// TIA Portal V17 export
// export: Created 2025-06-26T07:49:40.7746535Z, ExportSetting WithDefaults, DisplayName Totally Integrated Automation Portal, DisplayVersion V17 Update 8, DisplayName TIA Portal Openness, DisplayVersion V17 Update 8, DisplayName TIA Portal Version Control Interface, DisplayVersion V17, DisplayName STEP 7 Professional, DisplayVersion V17 Update 8, DisplayName STEP 7 Safety, DisplayVersion V17 Update 6, DisplayName WinCC Advanced, DisplayVersion V17 Update 8
FUNCTION_BLOCK "Evaluate"   // FB26, FBD
TITLE = Evaluate machine state conditions
{ S7_Optimized_Access := 'TRUE' }
AUTHOR : Heaten
VERSION : 0.1
// stored: AutoNumber true, IsIECCheckEnabled false, IsRetainMemResEnabled false, MemoryReserve 0, SetENOAutomatically false, UDAEnableTagReadback false
   VAR
      TOF2_StandbyPauseTime { S7_SetPoint := 'True'} : TOF_TIME;
      TON2_Standby { S7_SetPoint := 'True'} : TON_TIME;
      TON3_PrepareStart { S7_SetPoint := 'True'} : TON_TIME;
      TON4_Start { S7_SetPoint := 'True'} : TON_TIME;
      TON5_Warmup { S7_SetPoint := 'True'} : TON_TIME;
      TON7_Stop { S7_SetPoint := 'True'} : TON_TIME;
      MinimumPriming { S7_SetPoint := 'True'} : TON_TIME;
   END_VAR
   VAR_TEMP
      HydrolockSpeed : Real;
      HeatSinkTemperatureMax : Real;
   END_VAR
BEGIN

REGION Network 1: Check running condition: system initialized
   // Add more conditions here
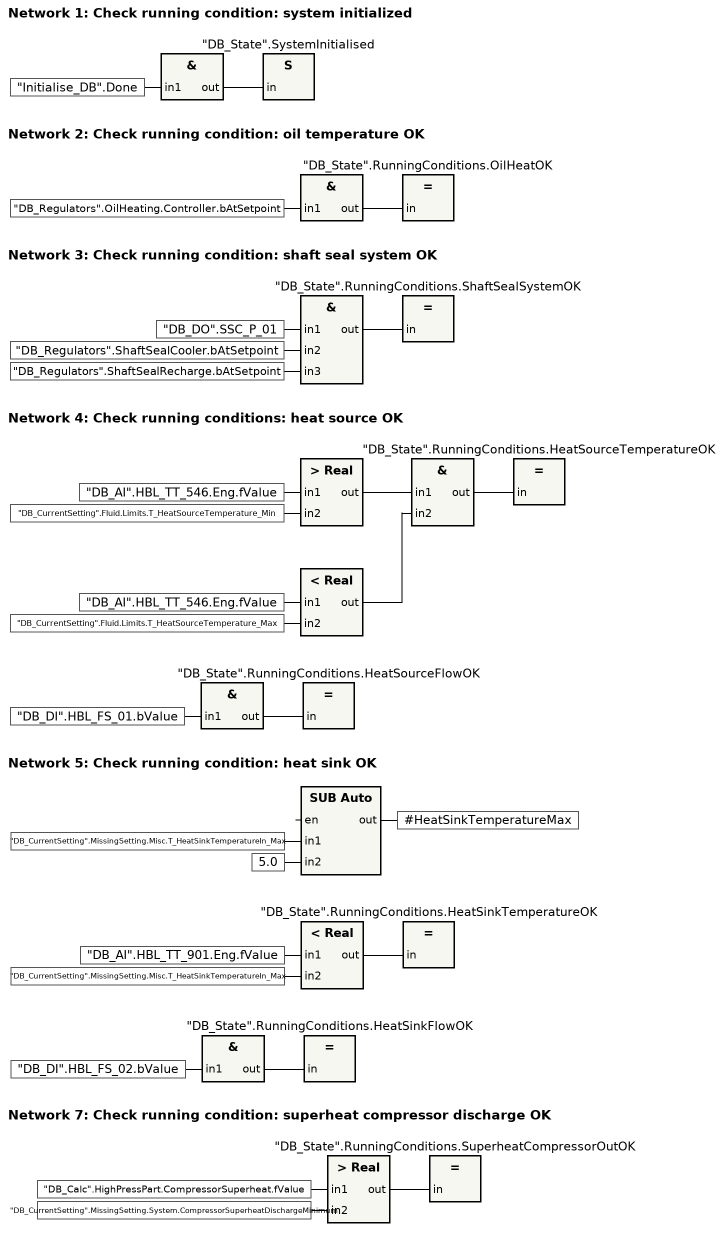
   IF "Initialise_DB".Done THEN "DB_State".SystemInitialised := TRUE; END_IF;
END_REGION

REGION Network 2: Check running condition: oil temperature OK
   "DB_State".RunningConditions.OilHeatOK := "DB_Regulators".OilHeating.Controller.bAtSetpoint;
END_REGION

REGION Network 3: Check running condition: shaft seal system OK
   "DB_State".RunningConditions.ShaftSealSystemOK := "DB_DO".SSC_P_01 AND "DB_Regulators".ShaftSealCooler.bAtSetpoint AND "DB_Regulators".ShaftSealRecharge.bAtSetpoint;
END_REGION

REGION Network 4: Check running conditions: heat source OK
   "DB_State".RunningConditions.HeatSourceTemperatureOK := ("DB_AI".HBL_TT_546.Eng.fValue > "DB_CurrentSetting".Fluid.Limits.T_HeatSourceTemperature_Min) AND ("DB_AI".HBL_TT_546.Eng.fValue < "DB_CurrentSetting".Fluid.Limits.T_HeatSourceTemperature_Max);
   "DB_State".RunningConditions.HeatSourceFlowOK := "DB_DI".HBL_FS_01.bValue;
END_REGION

REGION Network 5: Check running condition: heat sink OK
   // NOTE: leave a little headroom to the limit for standby, otherwise the machine shuts down (via alarm 2101) at the same temperature as it should go to standby on
   #HeatSinkTemperatureMax := "DB_CurrentSetting".MissingSetting.Misc.T_HeatSinkTemperatureIn_Max - 5.0;
   "DB_State".RunningConditions.HeatSinkTemperatureOK := "DB_AI".HBL_TT_901.Eng.fValue < "DB_CurrentSetting".MissingSetting.Misc.T_HeatSinkTemperatureIn_Max;
   "DB_State".RunningConditions.HeatSinkFlowOK := "DB_DI".HBL_FS_02.bValue;
END_REGION

REGION Network 6 (SCL): Check running condition: recuperator working
   // Recuperator sits between evaporator and compressor and SHOULD INCREASE THE SUPERHEAT (ie delta T over the recuperator should be positive)
   // 
   // Recuperator window: must add at least "DB_CurrentSetting".MissingSetting.System.RecuperatorSuperheatGainWorking degrees to be considered working, 
   // but can then fall as low as "DB_CurrentSetting".MissingSetting.System.RecuperatorSuperheatGainNotWorking degrees before it is considered not working again
   (*
   IF ("DB_Calc".LowPressPart.CompressorSuperheat.fValue - 2) <      //If the superheat at compressor inlet minus 2 is smaller than
       "DB_Calc".LowPressPart.EvaporatorSuperheat.fValue THEN          //the superheat at the evaporator, the recuperator doesn´t work
       "StateMachine_DB".RunningConditions.RecuperatorWorking := FALSE;
   ELSIF
       ("DB_Calc".LowPressPart.CompressorSuperheat.fValue + 3) >     //If the superheat at compressor inlet plus 3 is bigger than
       "DB_Calc".LowPressPart.EvaporatorSuperheat.fValue THEN          //the superheat at the evaporator, the recuperator works
       "StateMachine_DB".RunningConditions.RecuperatorWorking := TRUE;
   END_IF;
   *)

   // Rewritten with user-defined limits and right-side-up logic
   // Also don't evaluate the condition unless it's relevant, to avoid odd conditions during earlier states/cold start setting this accidentally
   IF "DB_State".State.State_Number = 5 OR "DB_State".State.State_Number = 6 THEN
       IF "DB_Calc".LowPressPart.CompressorSuperheat.fValue > "DB_Calc".LowPressPart.EvaporatorSuperheat.fValue + "DB_CurrentSetting".MissingSetting.System.RecuperatorDeltaTWorking THEN
           "DB_State".RunningConditions.RecuperatorWorking := TRUE;
       ELSIF "DB_Calc".LowPressPart.CompressorSuperheat.fValue < "DB_Calc".LowPressPart.EvaporatorSuperheat.fValue + "DB_CurrentSetting".MissingSetting.System.RecuperatorDeltaTNotWorking THEN
           "DB_State".RunningConditions.RecuperatorWorking := FALSE;
       END_IF;
   ELSE
       "DB_State".RunningConditions.RecuperatorWorking := FALSE;
   END_IF;
END_REGION

REGION Network 7: Check running condition: superheat compressor discharge OK
   "DB_State".RunningConditions.SuperheatCompressorOutOK := "DB_Calc".HighPressPart.CompressorSuperheat.fValue > "DB_CurrentSetting".MissingSetting.System.CompressorSuperheatDischargeMinimum;
END_REGION

REGION Network 8: Check running condition: at or above hydrolock speed
   // Give a small margin for error, so if it sits at, for example 288.2 RPM and the limit is 290, it will work.
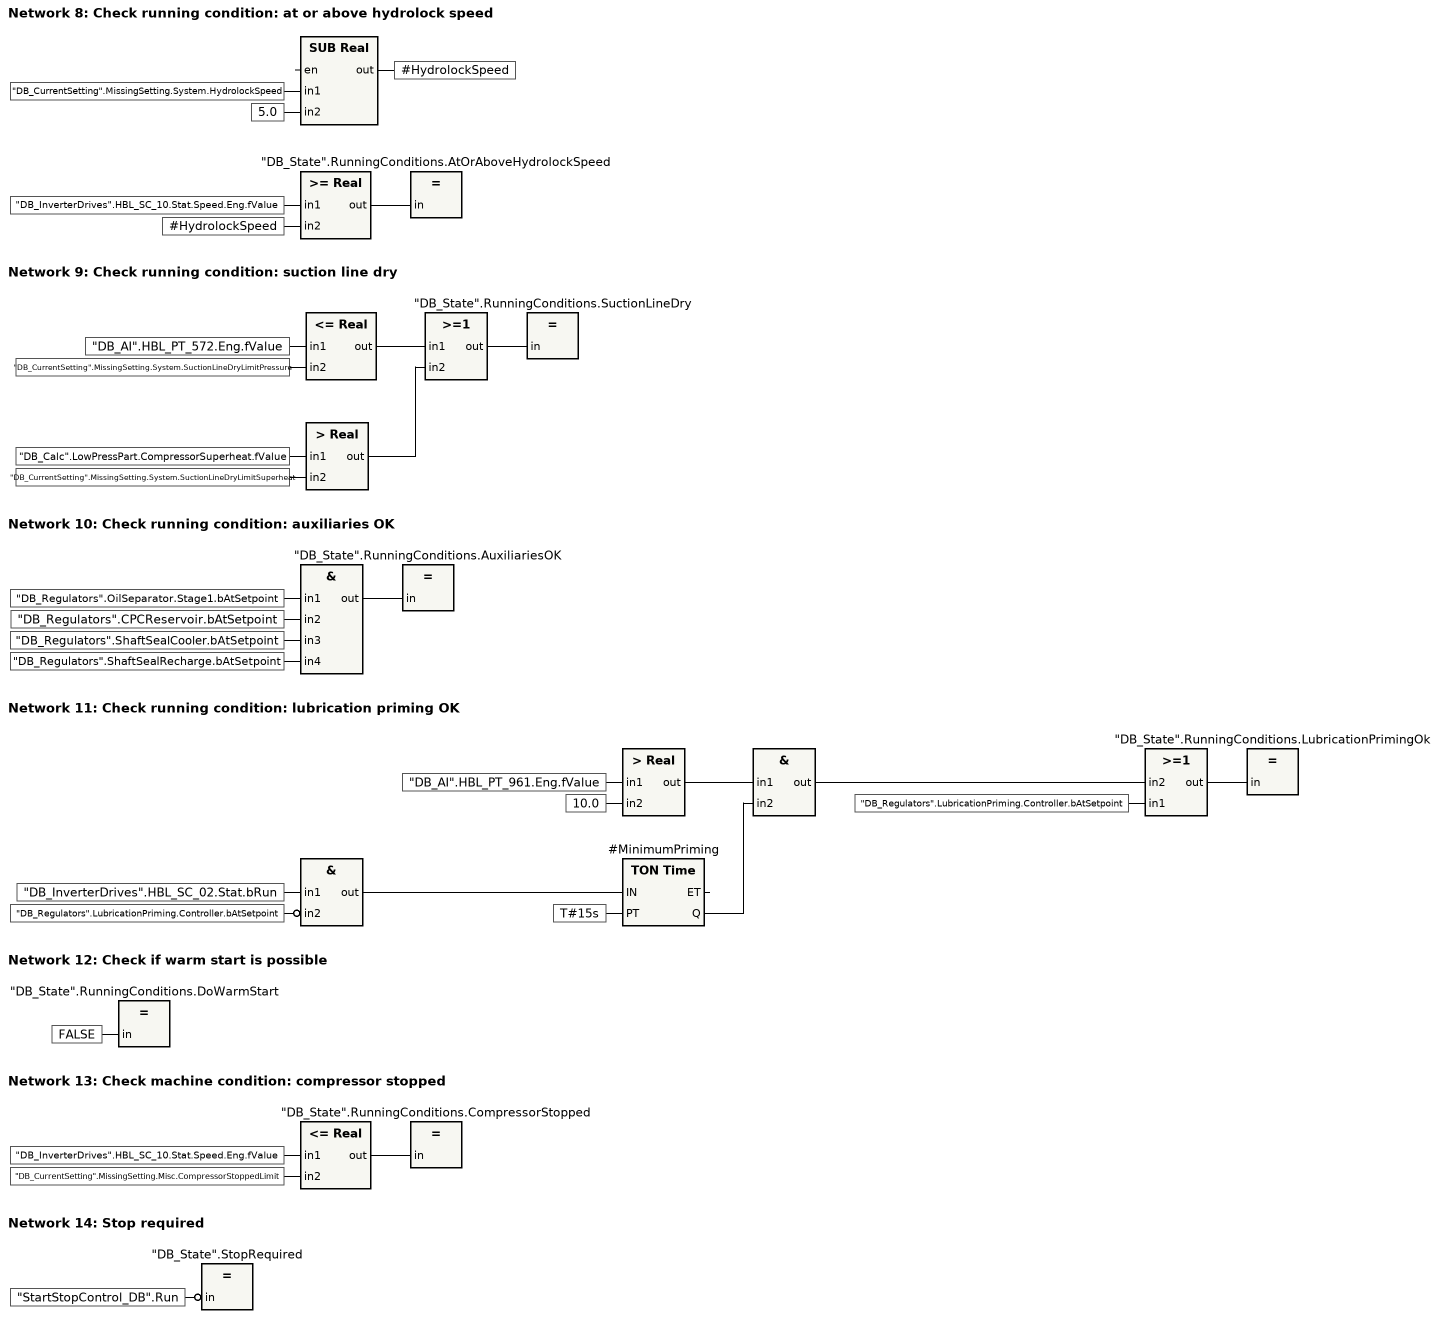
   #HydrolockSpeed := "DB_CurrentSetting".MissingSetting.System.HydrolockSpeed - 5.0;
   "DB_State".RunningConditions.AtOrAboveHydrolockSpeed := "DB_InverterDrives".HBL_SC_10.Stat.Speed.Eng.fValue >= #HydrolockSpeed;
END_REGION

REGION Network 9: Check running condition: suction line dry
   "DB_State".RunningConditions.SuctionLineDry := ("DB_AI".HBL_PT_572.Eng.fValue <= "DB_CurrentSetting".MissingSetting.System.SuctionLineDryLimitPressure) OR ("DB_Calc".LowPressPart.CompressorSuperheat.fValue > "DB_CurrentSetting".MissingSetting.System.SuctionLineDryLimitSuperheat);
END_REGION

REGION Network 10: Check running condition: auxiliaries OK
   "DB_State".RunningConditions.AuxiliariesOK := "DB_Regulators".OilSeparator.Stage1.bAtSetpoint AND "DB_Regulators".CPCReservoir.bAtSetpoint AND "DB_Regulators".ShaftSealCooler.bAtSetpoint AND "DB_Regulators".ShaftSealRecharge.bAtSetpoint;
END_REGION

REGION Network 11: Check running condition: lubrication priming OK
   // The simplest is to just look at the regulator's .bAtSetpoint bit. But the lubrication priming pump may be too small to reach the setpoint. So a hybrid condition is:
   // IF the pressure is at setpoint OR
   // the motor has been running for at least X sec when not at setpoint AND 
   // the developed lubrication pressure is greater than Y kPa THEN
   // the lubrication system is working ok.
   // NOTE: hardcoded params = bad!!
   #MinimumPriming(IN := "DB_InverterDrives".HBL_SC_02.Stat.bRun AND NOT "DB_Regulators".LubricationPriming.Controller.bAtSetpoint,   // TON
                   PT := T#15s);
   "DB_State".RunningConditions.LubricationPrimingOk := (("DB_AI".HBL_PT_961.Eng.fValue > 10.0) AND #MinimumPriming.Q) OR "DB_Regulators".LubricationPriming.Controller.bAtSetpoint;
END_REGION

REGION Network 12: Check if warm start is possible
   // Think of an appropriate condition
   "DB_State".RunningConditions.DoWarmStart := FALSE;
END_REGION

REGION Network 13: Check machine condition: compressor stopped
   "DB_State".RunningConditions.CompressorStopped := "DB_InverterDrives".HBL_SC_10.Stat.Speed.Eng.fValue <= "DB_CurrentSetting".MissingSetting.Misc.CompressorStoppedLimit;
END_REGION

REGION Network 14: Stop required
   // NOte: stop conditions are evaluated by FB30 StartStopControl
   "DB_State".StopRequired := NOT "StartStopControl_DB".Run;
END_REGION

REGION Network 15: Check for risk of hydrolock
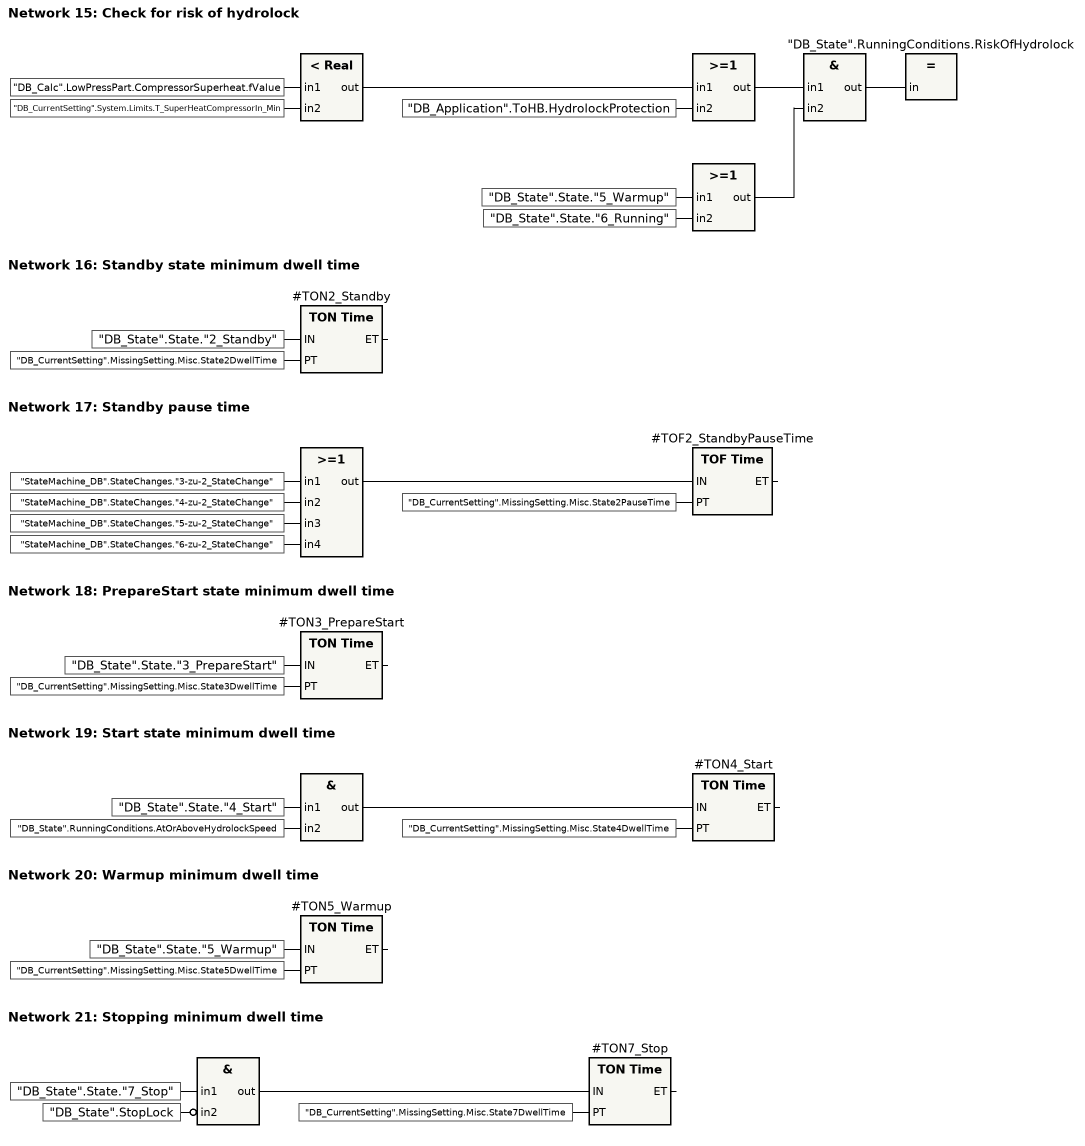
   "DB_State".RunningConditions.RiskOfHydrolock := (("DB_Calc".LowPressPart.CompressorSuperheat.fValue < "DB_CurrentSetting".System.Limits.T_SuperHeatCompressorIn_Min) OR "DB_Application".ToHB.HydrolockProtection) AND ("DB_State".State."5_Warmup" OR "DB_State".State."6_Running");
END_REGION

REGION Network 16: Standby state minimum dwell time
   #TON2_Standby(IN := "DB_State".State."2_Standby",   // TON
                 PT := "DB_CurrentSetting".MissingSetting.Misc.State2DwellTime);
END_REGION

REGION Network 17: Standby pause time
   // Minimum pause in Standby before resume
   #TOF2_StandbyPauseTime(IN := "StateMachine_DB".StateChanges."3-zu-2_StateChange" OR "StateMachine_DB".StateChanges."4-zu-2_StateChange" OR "StateMachine_DB".StateChanges."5-zu-2_StateChange" OR "StateMachine_DB".StateChanges."6-zu-2_StateChange",   // TOF
                          PT := "DB_CurrentSetting".MissingSetting.Misc.State2PauseTime);
END_REGION

REGION Network 18: PrepareStart state minimum dwell time
   #TON3_PrepareStart(IN := "DB_State".State."3_PrepareStart",   // TON
                      PT := "DB_CurrentSetting".MissingSetting.Misc.State3DwellTime);
END_REGION

REGION Network 19: Start state minimum dwell time
   #TON4_Start(IN := "DB_State".State."4_Start" AND "DB_State".RunningConditions.AtOrAboveHydrolockSpeed,   // TON
               PT := "DB_CurrentSetting".MissingSetting.Misc.State4DwellTime);
END_REGION

REGION Network 20: Warmup minimum dwell time
   #TON5_Warmup(IN := "DB_State".State."5_Warmup",   // TON
                PT := "DB_CurrentSetting".MissingSetting.Misc.State5DwellTime);
END_REGION

REGION Network 21: Stopping minimum dwell time
   #TON7_Stop(IN := "DB_State".State."7_Stop" AND NOT "DB_State".StopLock,   // TON
              PT := "DB_CurrentSetting".MissingSetting.Misc.State7DwellTime);
END_REGION
END_FUNCTION_BLOCK
